(* IEC 61131-3 sources: POMIRTS_lab3/AS/Library/MTPrintHW/V1.02.0, 3 files *)

(* ---- MTPrintHW.typ ---- *)
(********************************************************************
* COPYRIGHT -- Bernecker + Rainer
 ********************************************************************
 * Library: MTPrintHW
 * File: MTPrintHW.typ
 * Author: B&R
 ********************************************************************
 * Data types of library MTPrintHW
 ********************************************************************)
(*Types for MTPringHWRegMarkCapture*)

TYPE
	MTPrintHWRegMarkCaptureParaType : 	STRUCT
		PositionSource : USINT; (*Position, which should be latched on the drive.*)
		MeassuredEdge : USINT; (*Edge selection for the print mark trigger event.*)
		MinRegMarkWidth : REAL; (*Minimum width of a valid trigger event.*)
		MaxRegMarkWidth : REAL; (*Maximum width of a valid trigger event.*)
		ExpectionWindowWidth : REAL; (*Window in which the valid trigger signal can occur after/before the expected position. *)
		SetRegMarkPosition : REAL; (*Position where print mark is expected.*)
		SensorDelayTime : DINT; (*Registration mark sensor delay [µs].*)
	END_STRUCT;
	MTPrintHWRegMarkCaptInternalType : 	STRUCT
		Ts : REAL; (*Task cycle time. Units: [s].*)
		AxisModuloPosition : DINT; (*Data for internal use.*)
		EdgeDetectMastertimePosition : REAL; (*Data for internal use.*)
		EdgeDetectSlavetimePosition : REAL; (*Data for internal use.*)
		ParameterValid : BOOL; (*Data for internal use.*)
		AxisReference : REFERENCE TO UDINT; (*Data for internal use.*)
		Parameter : MTPrintHWRegMarkCaptureParaType; (*Data for internal use.*)
		State : USINT; (*Data for internal use.*)
		AxisFactor : DINT; (*Data for internal use.*)
		AxisPeriod : DINT; (*Data for internal use.*)
		MaxExpectionPosition : DINT; (*Data for internal use.*)
		MinExpectionPosition : DINT; (*Data for internal use.*)
		ActBufferIndex : UINT; (*Data for internal use.*)
		PositionBufferPointer : UDINT; (*Data for internal use.*)
		TimeBufferPointer : UDINT; (*Data for internal use.*)
		AxisSpeed : REAL; (*Data for internal use.*)
		AxisSystemTime : UDINT; (*Data for internal use.*)
		AxisUpdateTime : UDINT; (*Data for internal use.*)
		NumberOfOccuredWindows : UDINT; (*Data for internal use.*)
		EdgeDetectMastertimeOld : DINT; (*Data for internal use.*)
		LastSavedPosition : DINT; (*Data for internal use.*)
		InExpectionWindow : BOOL; (*Data for internal use.*)
		InExpectionWindowOld : BOOL; (*Data for internal use.*)
		FunctionBlockReadCyclicPosition : MC_BR_ReadCyclicPosition; (*Data for internal use.*)
		FunctionBlockCyclicDataInfo : MC_BR_CyclicReadDataInfo; (*Data for internal use.*)
		FunctionBlockCyclicRead : ARRAY[0..1]OF MC_BR_CyclicRead; (*Data for internal use.*)
		FunctionBlockReadParameter : ARRAY[0..1]OF MC_ReadParameter; (*Data for internal use.*)
		FunctionBlockMovingAverage : movAvg_typ; (*Data for internal use.*)
		ActRegMarkPositionErrorOld : REAL; (*Data for internal use.*)
		Update : BOOL; (*Data for internal use.*)
		UpdateOld : BOOL; (*Data for internal use.*)
		EnableOld : BOOL; (*Data for internal use.*)
		Bootkey : UDINT; (*Data for internal use.*)
		SystemTimeOld : UDINT; (*Data for internal use.*)
		ModuloPositionOld : DINT; (*Data for internal use.*)
	END_STRUCT;
	movAvg_typ : 	STRUCT
		enable : BOOL; (*Enable function block.*)
		window : UINT; (*Number of cycles used to generate the average value. Valid value range: base > 0.*)
		update : BOOL; (*Update parameters*)
		u : REAL; (*Input.*)
		status : UINT; (*Function block status message.*)
		y : REAL; (*Output value.*)
		internal : movAvg_internal_typ; (*Data for internal use.*)
	END_STRUCT;
	movAvg_internal_typ : 	STRUCT
		statusTxt : STRING[100]; (*Function block status message as message text.*)
		Ts : REAL; (*Task cycle time. Units: [s].*)
		paraValid : BOOL; (*Data for internal use.*)
		update : BOOL; (*Data for internal use.*)
		n : UINT; (*Data for internal use.*)
		sum : LREAL; (*Data for internal use.*)
		buffer : ARRAY[0..127]OF REAL; (*Data for internal use.*)
		pBuffer : UDINT; (*Data for internal use.*)
		i_act : UINT; (*Data for internal use.*)
		i_old : UINT; (*Data for internal use.*)
		base : UINT; (*Data for internal use.*)
		bufferLength : UINT; (*Data for internal use.*)
		bufferFull : BOOL; (*Data for internal use.*)
		memAllocated : BOOL; (*Data for internal use.*)
		update_old : BOOL; (*Data for internal use.*)
		enable_old : BOOL; (*Data for internal use.*)
		Bootkey : UDINT; (*Data for internal use.*)
	END_STRUCT;
END_TYPE

(*MTPrintHWGetAxisValues*)

TYPE
	MTPrintHWGetAxisValInternalType : 	STRUCT  (*Data for internal use.*)
		CycleTime : REAL; (*Data for internal use.*)
		Axis : UDINT; (*Data for internal use.*)
		FubState : USINT; (*Data for internal use.*)
		EnableOld : BOOL; (*Data for internal use.*)
		AxisNettime : UDINT; (*Data for internal use.*)
		AxisPosition : DINT; (*Data for internal use.*)
		AxisVelocity : REAL; (*Data for internal use.*)
		MC_BR_CyclicRead_Time : MC_BR_CyclicRead; (*Data for internal use.*)
		MC_BR_CyclicRead_Pos : MC_BR_CyclicRead; (*Data for internal use.*)
		MC_BR_CyclicRead_Vel : MC_BR_CyclicRead; (*Data for internal use.*)
	END_STRUCT;
END_TYPE

(*Types for MTPrintHWCalcTrigger*)

TYPE
	MTPrintHWCalcTriggerInternalType : 	STRUCT
		CycleTime : REAL; (*Data for internal use.*)
		ParameterValid : BOOL; (*Data for internal use.*)
		ImageLength : DINT; (*Data for internal use.*)
		ImageOffset : DINT; (*Data for internal use.*)
		EnableOld : BOOL; (*Data for internal use.*)
		UpdateOld : BOOL; (*Data for internal use.*)
		AxisNettime : UDINT; (*Data for internal use.*)
		AxisPosition : DINT; (*Data for internal use.*)
		AxisVelocity : REAL; (*Data for internal use.*)
		AxisAcc : REAL; (*Data for internal use.*)
		TriggerPosition : DINT; (*Data for internal use.*)
		TriggerTime : UDINT; (*Data for internal use.*)
		LastTriggerTime : UDINT; (*Data for internal use.*)
		DeltaPosition : DINT; (*Data for internal use.*)
		DeltaTime : REAL; (*Data for internal use.*)
	END_STRUCT;
END_TYPE

(*Types for MTPrintHWTimeToPosition*)

TYPE
	MTPrintHWTimeToPosInternalType : 	STRUCT
		CycleTime : REAL; (*Data for internal use.*)
		ParameterValid : BOOL; (*Data for internal use.*)
		ActivatedEdge : ARRAY[0..39]OF BOOL; (*Data for internal use.*)
		EnableOld : BOOL; (*Data for internal use.*)
		UpdateOld : BOOL; (*Data for internal use.*)
		Record : BOOL; (*Data for internal use.*)
		StartRecordOld : BOOL; (*Data for internal use.*)
		AxisNettime : UDINT; (*Data for internal use.*)
		AxisPosition : DINT; (*Data for internal use.*)
		AxisPositionOld : DINT; (*Data for internal use.*)
		PositionCounter : UINT; (*Data for internal use.*)
		Time : UDINT; (*Data for internal use.*)
		Position : DINT; (*Data for internal use.*)
		pTime : REFERENCE TO UDINT; (*Data for internal use.*)
		pPosition : REFERENCE TO DINT; (*Data for internal use.*)
	END_STRUCT;
END_TYPE

(* ---- MTPrintHW.fun ---- *)
(********************************************************************
 * COPYRIGHT -- Bernecker + Rainer
 ********************************************************************
 * Library: MTPrintHW
 * File: MTPrintHW.fun
 * Author: B&R
 ********************************************************************
 * Functions and function blocks of library MTPrintHW
 ********************************************************************)

FUNCTION_BLOCK MTPrintHWRegMarkCapture (*Registration mark detection.*)
	VAR_INPUT
		Axis : UDINT; (*Axis reference for the axis on which registration mark detection is running.*)
		Enable : BOOL; (*Enable function block.*)
		Parameter : MTPrintHWRegMarkCaptureParaType; (*Registration mark parameters.*)
		MovingWindowLength : USINT; (*Number of values used to generate the average position error.*)
		Update : BOOL; (*Parameter update trigger.*)
		EdgeDetectSlavetime : DINT; (*Net time of slave (first) edge.*)
		EdgeDetectMastertime : DINT; (*Net time of master (last) edge.*)
		SearchRegMark : BOOL; (*Search for any registration mark with correct size.*)
	END_VAR
	VAR_OUTPUT
		Active : BOOL; (*Function block is active.*)
		Error : BOOL; (*Indicates an error.*)
		StatusID : DINT; (*Status information.*)
		UpdateDone : BOOL; (*Update done.*)
		ActRegMarkPosition : REAL; (*Currently measured position of the registration mark within one revolution.*)
		ActRegMarkPositionError : REAL; (*Absolute deviation between expected position ("RegMarkPosition") and measured position of the registration mark ("ActPosition") within one revolution.*)
		ActRegMarkSize : REAL; (*Actual size of detected registration mark.*)
		ValidRegMarks : UDINT; (*The number of valid trigger signals.*)
		MissedRegMarks : UDINT; (*The number of "missed" triggers (set to 0, after a valid trigger signal was detected again).*)
		AverageRegMarkPositionError : REAL; (*Average value of the last measured position errors.*)
	END_VAR
	VAR
		Internal : MTPrintHWRegMarkCaptInternalType; (*Data for internal use.*)
	END_VAR
END_FUNCTION_BLOCK

FUNCTION_BLOCK MTPrintHWGetAxisValues (*TODO: Add your comment here*) (*$GROUP=User*)
	VAR_INPUT
		Axis : UDINT; (*Axis reference.*)
		Enable : BOOL; (*Enable function block.*)
	END_VAR
	VAR_OUTPUT
		Active : USINT; (*Function block is active.*)
		Busy : USINT; (*Function block is*)
		Error : USINT; (*Indicates an error.*)
		StatusID : DINT; (*Status information.*)
		AxisNettime : UDINT; (*Axis nettime.*)
		AxisPosition : DINT; (*Axis position.*)
		AxisVelocity : REAL; (*Axus Velocity.*)
	END_VAR
	VAR
		Internal : MTPrintHWGetAxisValInternalType; (*Data for internal use.*)
	END_VAR
END_FUNCTION_BLOCK

FUNCTION_BLOCK MTPrintHWCalcTrigger
	VAR_INPUT
		Enable : BOOL; (*Enable function block.*)
		ImageLength : DINT; (*Length of Image.*)
		ImageOffset : DINT; (*Trigger position.*)
		Update : BOOL; (*Parameter update.*)
		AxisNettime : UDINT; (*Axis nettime.*)
		AxisPosition : DINT; (*Axis position.*)
		AxisVelocity : REAL; (*Axus Velocity.*)
	END_VAR
	VAR_OUTPUT
		Active : BOOL; (*Function block is active.*)
		Error : BOOL; (*Indicates an error.*)
		StatusID : DINT; (*Status information.*)
		UpdateDone : BOOL; (*Update done.*)
		TriggerTime : UDINT; (*Nettime for trigger.*)
		TriggerPosition : DINT; (*Position of trigger.*)
		LastTriggerTime : UDINT; (*Nettime of the last trigger.*)
	END_VAR
	VAR
		Internal : MTPrintHWCalcTriggerInternalType; (*Data for internal use.*)
	END_VAR
END_FUNCTION_BLOCK

FUNCTION_BLOCK MTPrintHWTimeToPosition
	VAR_INPUT
		Enable : BOOL; (*Enable function block.*)
		ActivatedEdge : ARRAY[0..39] OF BOOL; (*Activated edge for position calculation.*)
		Update : BOOL; (*Parameter update.*)
		EdgeTime : ARRAY[0..39] OF UDINT; (*Time for position calculation.*)
		AxisNettime : UDINT; (*Time.*)
		AxisPosition : DINT; (*Position.*)
		StartRecord : BOOL; (*Start Record Time and Position.*)
	END_VAR
	VAR_OUTPUT
		Active : BOOL; (*Function block is active.*)
		Error : BOOL; (*Indicates an error.*)
		StatusID : DINT; (*Status information.*)
		UpdateDone : BOOL; (*Update done.*)
		EdgePosition : ARRAY[0..39] OF DINT; (*Calculated position.*)
		NewPosition : BOOL; (*New position.*)
	END_VAR
	VAR
		Internal : MTPrintHWTimeToPosInternalType; (*Data for internal use.*)
	END_VAR
END_FUNCTION_BLOCK

(* ---- MTPrintHW.var ---- *)
(********************************************************************
 * COPYRIGHT -- Bernecker + Rainer
 ********************************************************************
 * Library: MTPrintHW
 * File: MTPrintHW.var
 * Author: B&R
 ********************************************************************
 * Constants of library MTPrintHW
 ********************************************************************)
VAR CONSTANT
	mtPRN_ERR_CYCLIC_READ : DINT := -1058006184; (*Error: MC_Cyclic_Read *)
	mtPRN_ERR_MEMORY : DINT := -1058006183; (*Error: An error occurred during memory allocation.*)
	mtPRN_ERR_IMAGE_LENGTH : DINT := -1058006182; (*Error: Image length invalid*)
	mtPRN_ERR_IMAGE_OFFSET : DINT := -1058006181; (*Error: Image offset invalid.*)
	mtPRN_ERR_LESS_POSITION : DINT := -1058006180; (*Error: Not enough position values.*)
	mtPRN_ERR_PARAMETER_INVALID : DINT := -1058006179; (*Error: One or more parameters higher or equal than one period.*)
	mtPRN_ERR_WIDTH_INVALID : DINT := -1058006178; (*Error: Defined print mark width invalid.*)
	mtPRN_ERR_WINDOW_INVALID : DINT := -1058006177; (*Error: Definded expection window invalid.*)
	mtPRN_ERR_NO_PERIOD : DINT := -1058006176; (*Error: Axis is not periodic.*)
	mtPRN_ERR_SENSOR_DELAY : DINT := -1058006175; (*Error: Sensor delay less than 0.*)
	mtPRN_WRN_IMAGE_LENGTH : DINT := -2131748008; (*Warning: Image length invalid*)
	mtPRN_WRN_IMAGE_OFFSET : DINT := -2131748007; (*Warning: Image offset invalid.*)
	mtPRN_WRN_WIDTH_INVALID : DINT := -2131748006; (*Warning: Defined print mark width invalid - kept last valid values.*)
	mtPRN_WRN_WINDOW_INVALID : DINT := -2131748005; (*Warning: Definded expection window invalid - kept last valid values.*)
	mtPRN_WRN_BUFFER_FULL : DINT := -2131748004; (*Warning: Internal buffer is full.*)
	mtPRN_WRN_SENSOR_DELAY : DINT := -2131748003; (*Warning: Sensor delay less than 0 - kept last valid values.*)
END_VAR
